(* IEC 61131-3 sources: Lasal/CPU_5344_V01/Class/cntrDistance, 1 file *)

(* ---- cntrDistance.st ---- *)
(*!
<Class
	Name               = "cntrDistance"
	Revision           = "0.0"
	RealtimeTask       = "false"
	CyclicTask         = "false"
	BackgroundTask     = "true"
	DefBackground      = "100 ms"
	Sigmatek           = "false"
	OSInterface        = "false"
	HighPriority       = "false"
	Automatic          = "false"
	UpdateMode         = "Prescan"
	SharedCommandTable = "true"
	Objectsize         = "(284,120)">
	<Channels>
		<Server Name="actPos" Visualized="false" Initialize="false" WriteProtected="false" Retentive="false"/>
		<Server Name="ClassSvr" Visualized="false" Initialize="false" WriteProtected="true" Retentive="false"/>
		<Server Name="resetSoftCounter" Visualized="true" Initialize="false" WriteProtected="false" Retentive="false"/>
		<Server Name="softCounter" Visualized="true" Initialize="false" WriteProtected="false" Retentive="SRam"/>
		<Server Name="totalCounter" Visualized="true" Initialize="false" WriteProtected="false" Retentive="SRam"/>
	</Channels>
</Class>
*)
cntrDistance : CLASS
  //Servers:
	ClassSvr 	: SvrChCmd_DINT;
	actPos 	: SvrCh_DINT;
	softCounter 	: SvrCh_DINT;
	totalCounter 	: SvrCh_DINT;
	resetSoftCounter 	: SvrCh_DINT;
  //Clients:
  //Variables:
		tmpCounter 	: DINT;
		timeWritten 	: UDINT;
		oldActPos 	: DINT;
		tmpDistance 	: DINT;
		tmpPos 	: DINT;
  //Functions:

	FUNCTION VIRTUAL GLOBAL Init;

	FUNCTION VIRTUAL GLOBAL Background
		VAR_INPUT
			EAX 	: UDINT;
		END_VAR
		VAR_OUTPUT
			state (EAX) 	: UDINT := READY;
		END_VAR;

	FUNCTION storeIt;

	FUNCTION VIRTUAL GLOBAL resetSoftCounter::Write
		VAR_INPUT
			input (EAX) 	: DINT;
		END_VAR
		VAR_OUTPUT
			result (EAX) 	: DINT;
		END_VAR;
  //Tables:
	FUNCTION @STD
		VAR_OUTPUT
			ret_code	: CONFSTATES;
		END_VAR;
	FUNCTION GLOBAL TAB @CT_;
END_CLASS;

// JdK 21-11-2019: class to count distance, they are stored in ram servers, don't write them to often
// every 1/10 mm change is handled, every 1 meter is counted, every 10m is stored, or every 5 minutes

FUNCTION VIRTUAL GLOBAL cntrDistance::Init

  tmpCounter:= totalCounter;
  timeWritten:= ops.tAbsolute;

END_FUNCTION

FUNCTION VIRTUAL GLOBAL cntrDistance::Background
	VAR_INPUT
		EAX 	: UDINT;
	END_VAR
	VAR_OUTPUT
		state (EAX) 	: UDINT;(* := READY *)
	END_VAR

  tmpPos:= abs(oldActPos-actPos);
  IF tmpPos > 10 THEN //don't handle the very small changes
    IF tmpPos < 10000 THEN //else, to big change, just ignore
      tmpDistance+= abs(oldActPos- actPos);
      IF tmpDistance > 10000 THEN //one meter
        totalCounter+= 1;
        softCounter+= 1;
        tmpDistance-= 10000;
        IF totalCounter-tmpCounter > 10 THEN
          storeIt();
        END_IF;
      END_IF;
    END_IF;
    oldActPos:= actPos;
  END_IF;

  IF totalCounter= tmpCounter THEN
    timeWritten:= ops.tAbsolute; //no need to write again
  ELSIF ops.tAbsolute-timeWritten > 300000 THEN //after 5 minutes
    storeIt();
  END_IF;

END_FUNCTION

FUNCTION VIRTUAL GLOBAL cntrDistance::resetSoftCounter::Write
	VAR_INPUT
		input (EAX) 	: DINT;
	END_VAR
	VAR_OUTPUT
		result (EAX) 	: DINT;
	END_VAR

	resetSoftCounter := input;
  softCounter:= 0;
  softCounter.Write(input:=softCounter);
	result := resetSoftCounter;

END_FUNCTION

FUNCTION cntrDistance::storeIt

  tmpCounter:=totalCounter;
  softCounter-= 1; //we can only store a new value
  totalCounter-= 1;
  softCounter.Write(input:=softCounter+1); //write action to store value
  totalCounter.Write(input:=totalCounter+1);

END_FUNCTION
